// TIA Portal project "Nastro_discesa" (V16)

(* hardware
DEVICE "S7-1200 station_1"  S7-1200 Station
   slot 0: "Telaio di montaggio_0"  S7-1200 Rack  Rack  V1.0
   slot 1: "PLC_1"  CPU 1215C DC/DC/Rly  6ES7 215-1HG40-0XB0  V4.2
*)

// ===== PLC "PLC_1"  CPU 1215C DC/DC/Rly =====

DATA_BLOCK "Blocco_dati_HMI"   // DB1
{ S7_Optimized_Access := 'TRUE' }
VERSION : 0.1
   VAR
      Jog_start : Bool;
      Jog_ripristino : Bool;
      "Passo 0" : Bool;
      "Passo 1" : Bool;
      "Passo 2" : Bool;
      "Passo 3" : Bool;
      "Passo 4" : Bool;
      "Passo 5" : Bool;
   END_VAR
BEGIN
END_DATA_BLOCK

FUNCTION "Ripristino" : Void   // FC1, LAD
{ S7_Optimized_Access := 'TRUE' }
VERSION : 0.1
BEGIN

REGION Network 1
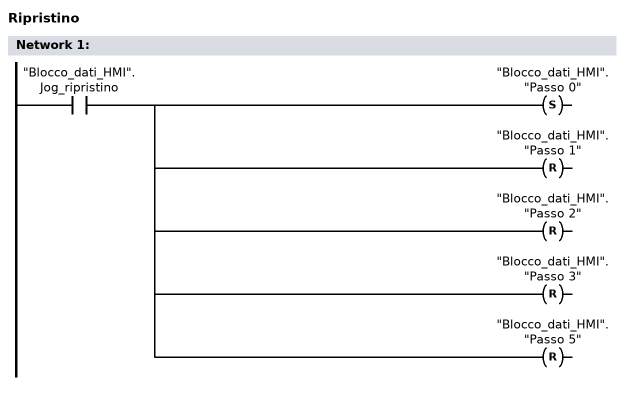
   RUNG wire#powerrail
      Contact( "Blocco_dati_HMI".Jog_ripristino )
      wire#w1
      S_Coil( "Blocco_dati_HMI"."Passo 0" )
   END_RUNG
   RUNG wire#w1
      R_Coil( "Blocco_dati_HMI"."Passo 1" )
   END_RUNG
   RUNG wire#w1
      R_Coil( "Blocco_dati_HMI"."Passo 2" )
   END_RUNG
   RUNG wire#w1
      R_Coil( "Blocco_dati_HMI"."Passo 3" )
   END_RUNG
   RUNG wire#w1
      R_Coil( "Blocco_dati_HMI"."Passo 5" )
   END_RUNG
   // the same network as SCL:
   IF "Blocco_dati_HMI".Jog_ripristino THEN
       "Blocco_dati_HMI"."Passo 0" := TRUE;
       "Blocco_dati_HMI"."Passo 1" := FALSE;
       "Blocco_dati_HMI"."Passo 2" := FALSE;
       "Blocco_dati_HMI"."Passo 3" := FALSE;
       "Blocco_dati_HMI"."Passo 5" := FALSE;
   END_IF;
END_REGION
END_FUNCTION

FUNCTION "Struttura_dei_passi" : Void   // FC2, LAD
{ S7_Optimized_Access := 'TRUE' }
VERSION : 0.1
BEGIN
END_FUNCTION

FUNCTION "Attivazione_delle_uscite" : Void   // FC3, LAD
{ S7_Optimized_Access := 'TRUE' }
VERSION : 0.1
BEGIN
END_FUNCTION

ORGANIZATION_BLOCK "Main"   // OB1, LAD, ProgramCycle
TITLE = "Main Program Sweep (Cycle)"
{ S7_Optimized_Access := 'TRUE' }
VERSION : 0.1
   VAR_INPUT
      Initial_Call : Bool;   // Initial call of this OB
      Remanence : Bool;   // =True, if remanent data are available
   END_VAR
BEGIN

REGION Network 1
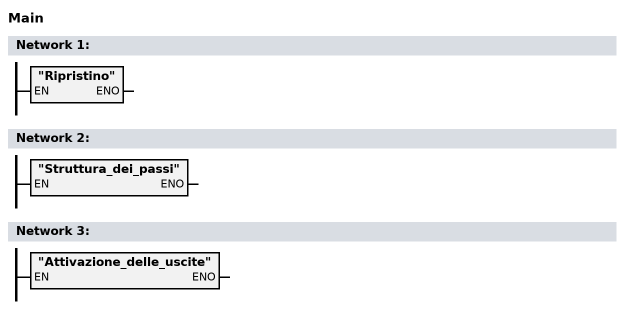
   RUNG wire#powerrail
      "Ripristino"()
   END_RUNG
   // the same network as SCL:
   "Ripristino"();
END_REGION

REGION Network 2
   RUNG wire#powerrail
      "Struttura_dei_passi"()
   END_RUNG
   // the same network as SCL:
   "Struttura_dei_passi"();
END_REGION

REGION Network 3
   RUNG wire#powerrail
      "Attivazione_delle_uscite"()
   END_RUNG
   // the same network as SCL:
   "Attivazione_delle_uscite"();
END_REGION
END_ORGANIZATION_BLOCK